Fanuc KAREL source: KT00779.KL

PROGRAM KT00779
%NOLOCKGROUP
VAR
  H1: ARRAY[2] OF SHORT
  H2: ARRAY[2] OF SHORT
  OUT: REAL
BEGIN
  H1[1] = 2
  H2[1] = 3
  H1[1] = 2
  H2[1] = 3
  OUT = ASIN(H1[1])
END KT00779
